// TIA Portal V20 export
FUNCTION_BLOCK "FB_ChillerSMC"   // FB541, SCL
{ S7_Optimized_Access := 'TRUE' }
// stored: AutoNumber false, MemoryReserve 100, SetENOAutomatically false
   VAR
      sTimeHeadChillerCutOff { S7_SetPoint := 'True'} : TON_TIME;
      sTimeHeadChillerTemperature { S7_SetPoint := 'True'} : TON_TIME;
      sTimeSourceChillerCutOff { S7_SetPoint := 'True'} : TON_TIME;
      sTimeSourceChillerTemperature { S7_SetPoint := 'True'} : TON_TIME;
   END_VAR
   VAR CONSTANT
      TIME_CHILLER_CUTOFF : Time := T#8s;
      TIME_CHILLER_TEMPERATURE : Time := T#8s;
   END_VAR
BEGIN
   REGION Description header 
       //==================================================================================
       // POSALUX Swiss SA / (C) Copyright 2025
       //----------------------------------------------------------------------------------
       // Title: FB_Chiller_SMC
       // Comment/Function:
       // Author: Fabien Waldt
       // Engineering: TIA Portal v19
       //----------------------------------------------------------------------------------
       // Change log table:
       // Version  | Date     | Expert in charge | Changes applied
       // ---------|----------|------------------|------------------------------------
       // 00.00.01 | 20250904 | FWA              | First released version
       // ==================================================================================
   END_REGION

   REGION Head Chiller
       REGION Alarm Head Chiller : CutOff
           #sTimeHeadChillerCutOff(IN := "DB_PowerOn".sMachineReadySoft AND NOT "DB_DigitalInputs".sHeadChillerCutOff.sSWStatus,
                                   PT := #TIME_CHILLER_CUTOFF,
                                   Q => "LBP_AlarmMsgs".UserA[02].A70UUxx[28]);
       END_REGION

       REGION Alarm Head Chiller : Temperature
           #sTimeHeadChillerTemperature(IN := "DB_PowerOn".sMachineReadySoft AND NOT "DB_DigitalInputs".sHeadChillerTemperature.sSWStatus,
                                        PT := #TIME_CHILLER_TEMPERATURE,
                                        Q => "LBP_AlarmMsgs".UserA[02].A70UUxx[29]);
       END_REGION
   END_REGION

   REGION Source Chiller
       REGION Alarm Source Chiller : CutOff
           #sTimeSourceChillerCutOff(IN := "DB_PowerOn".sMachineReadySoft AND NOT "DB_DigitalInputs".sSourceChillerCutOff.sSWStatus,
                                     PT := #TIME_CHILLER_CUTOFF,
                                     Q => "LBP_AlarmMsgs".UserA[02].A70UUxx[30]);
       END_REGION

       REGION Alarm Source Chiller : Temperature
           #sTimeSourceChillerTemperature(IN := "DB_PowerOn".sMachineReadySoft AND NOT "DB_DigitalInputs".sSourceChillerTemperature.sSWStatus,
                                          PT := #TIME_CHILLER_TEMPERATURE,
                                          Q => "LBP_AlarmMsgs".UserA[02].A70UUxx[31]);
       END_REGION
   END_REGION
END_FUNCTION_BLOCK
